PROGRAM PRG_06_HomePosition
VAR
	iStepHome: INT;
	SR_MachineHoming: SR;
	R_TRIG_MachineHoming: R_TRIG;	
	TON_HomingStep10: TON;
END_VAR

VAR PERSISTENT
	
END_VAR

	IF		NOT bSafetyOK OR IN_FaultReset OR bAutoCrossCut OR bTurretReturn OR NOT SR_MachineHoming.Q1
	THEN	iStepHome	:=	0;
			bMachineHoming := FALSE;
	END_IF
	
			R_TRIG_MachineHoming(	CLK:= IN_bLiftingPosition AND NOT bTurretReturn AND NOT bAutoCrossCut AND NOT OUT_bSawOn,
									Q=> );	
			SR_MachineHoming(	SET1:= R_TRIG_MachineHoming.Q AND NOT SR_MachineHoming.Q1,
								RESET:= (R_TRIG_MachineHoming.Q AND SR_MachineHoming.Q1) OR NOT bSafetyOK OR IN_FaultReset, 
								Q1=> );
	
IF bMachineHoming THEN
	OUT_bLiftingPositionLED := TRUE ;
ELSE
	OUT_bLiftingPositionLED := FALSE ;
END_IF

CASE iStepHome OF
	0:	// Init step
		bTurretHome		:= FALSE; 
	    bCarriageHomeLH	:= FALSE;
	    bCarriageHomeRH	:= FALSE;
	    bCrossCutHomeLH	:= FALSE;
	    bCrossCutHomeRH	:= FALSE;
		bZAxisHome := FALSE;
		TON_HomingStep10.IN := FALSE;
	
		IF R_TRIG_MachineHoming.Q AND bSafetyOK AND NOT OUT_bSawOn THEN
			bMachineHoming := TRUE ;
			iStepHome := 5 ;
		ELSE
			bMachineHoming := FALSE ;
		END_IF
		
	5:	// Raise Z-axis all the way up
	
		IF IN_bSawUpLimit AND bSafetyOK AND bMachineHoming THEN
			bZAxisHome := TRUE ;
		ELSE
			bZAxisHome := FALSE ; 
			iStepHome := 7 ;
		END_IF
		
	7:	// Move crosscut motor to centre
	 
		IF IN_uCrossCutSSI < (uRailLimitLeft + uRailLimitRight)/2 AND bSafetyOK AND bMachineHoming THEN
			bCrossCutHomeLH := TRUE ;
			bCrossCutHomeRH := FALSE ;
		ELSIF IN_uCrossCutSSI > (uRailLimitLeft + uRailLimitRight)/2 AND bSafetyOK AND bMachineHoming THEN
			bCrossCutHomeRH := TRUE ;
			bCrossCutHomeLH := FALSE ;
		ELSIF (IN_uCrossCutSSI > ((uRailLimitLeft + uRailLimitRight)/2) - 50) OR (IN_uCrossCutSSI < ((uRailLimitLeft + uRailLimitRight)/2) + 50) AND bSafetyOK AND bMachineHoming THEN
			bCrossCutHomeLH := FALSE ;
			bCrossCutHomeRH := FALSE ;
			iStepHome := 10 ;
		END_IF
	
	10:	// Rotate turret to max -90°
	
			TON_HomingStep10(IN:= , PT:= T#1S, Q=> , ET=> );
		IF NOT bTurretCCW AND bSafetyOK AND bMachineHoming THEN
			bTurretHome := TRUE ;
		ELSIF bTurretCCW AND bSafetyOK AND bMachineHoming THEN
			TON_HomingStep10.IN := TRUE ;
			bTurretHome := FALSE ;
			IF TON_HomingStep10.Q THEN
			    iStepHome := 20 ;
			END_IF
			
		END_IF
	
	20: // Offset carriage a little to the right		// 32.3 < CarriageHome < 32.5
	
		IF (fbCarriagePOS.Out.rScaled < 32.3) AND bMachineHoming AND bSafetyOK THEN
			bCarriageHomeRH := TRUE ;
			bCarriageHomeLH := FALSE ;
		ELSIF (fbCarriagePOS.Out.rScaled > 32.5) AND bMachineHoming AND bSafetyOK THEN
			bCarriageHomeLH := TRUE ;
			bCarriageHomeRH := FALSE ;
		ELSIF (fbCarriagePOS.Out.rScaled > 32.3) AND (fbCarriagePOS.Out.rScaled < 32.5) THEN
			bCarriageHomeRH := FALSE ;
			bCarriageHomeLH := FALSE ;
			iStepHome := 30 ;
		END_IF
	
	30: //Crosscut offset towards the control panel (CUT direction)		// 55.5 < CrosscutHome < 55.75
	
		IF (fbCrosscutSSI.Out.rScaled < 55.5) AND bMachineHoming AND bSafetyOK THEN
			bCrossCutHomeLH := TRUE ;
			bCrossCutHomeRH := FALSE ;
		ELSIF (fbCrosscutSSI.Out.rScaled > 55.75) AND bMachineHoming AND bSafetyOK THEN
			bCrossCutHomeRH := TRUE ;
			bCrossCutHomeLH := FALSE ;
		ELSIF (fbCrosscutSSI.Out.rScaled > 55.5) AND (fbCrosscutSSI.Out.rScaled < 55.75) THEN
			bCrossCutHomeLH := FALSE ;
			bCrossCutHomeRH := FALSE ;
			iStepHome := 0 ;
		END_IF
		
END_CASE

END_PROGRAM

(* stored: Version 1.1.0.1, ProductVersion 3.1.4024.12
   POU PRG_06_HomePosition: Id {e66157ee-61e1-4e85-a7d7-00daf40c8d31}, SpecialFunc None *)
